KUKA KRL data list: CK1STXXX.dat

&ACCESS RVP
&REL 2
&PARAM EDITMASK = *
DEFDAT  CK1STXXX
;FOLD EXTERNAL DECLARATIONS;%{PE}%MKUKATPBASIS,%CEXT,%VCOMMON,%P
;FOLD BASISTECH EXT;%{PE}%MKUKATPBASIS,%CEXT,%VEXT,%P
EXT  BAS (BAS_COMMAND  :IN,REAL  :IN )
DECL INT SUCCESS
;ENDFOLD (BASISTECH EXT)
;FOLD USER EXT;%{E}%MKUKATPUSER,%CEXT,%VEXT,%P
;Make here your modifications

;ENDFOLD (USER EXT)
;ENDFOLD (EXTERNAL DECLARATIONS)
DECL E6POS XTag7={X -521.268,Y 1581.23206,Z 8.80100,A 49.4600,B 19.4680,C 176.878,S 6,T 59,E1 0.0,E2 0.0,E3 0.0,E4 0.0,E5 0.0,E6 0.0}
DECL FDAT FTag7={TOOL_NO 1,BASE_NO 0,IPO_FRAME #BASE}
DECL PDAT PPDAT1={VEL 80.0000,ACC 100.000,APO_DIST 0.0}
DECL E6POS XTag1={X -521.268,Y 1620.44702,Z -535.910,A 49.4600,B 19.4680,C 176.878,S 6,T 59,E1 0.0,E2 0.0,E3 0.0,E4 0.0,E5 0.0,E6 0.0}
DECL FDAT FTag1={TOOL_NO 1,BASE_NO 0,IPO_FRAME #BASE}
DECL PDAT PPDAT2={VEL 80.0000,ACC 100.000,APO_DIST 100.000}
DECL E6POS XTag2={X -534.322,Y 1875.80,Z -416.009,A 69.9700,B -0.00600000,C 179.993,S 6,T 59,E1 0.0,E2 0.0,E3 0.0,E4 0.0,E5 0.0,E6 0.0}
DECL FDAT FTag2={TOOL_NO 1,BASE_NO 0,IPO_FRAME #BASE}
DECL PDAT PPDAT3={VEL 80.0000,ACC 100.000,APO_DIST 50.0000}
DECL E6POS XTag3={X -534.339,Y 1875.79297,Z -303.179,A 69.9700,B -0.00600000,C 179.993,S 6,T 59,E1 0.0,E2 0.0,E3 0.0,E4 0.0,E5 0.0,E6 0.0}
DECL FDAT FTag3={TOOL_NO 1,BASE_NO 0,IPO_FRAME #BASE}
DECL LDAT LCPDAT1={VEL 0.800000,ACC 100.000,APO_DIST 0.0,APO_FAC 50.0000}
DECL E6POS XTag4={X -534.322,Y 1875.80,Z -416.008,A 69.9700,B -0.00600000,C 179.993,S 6,T 59,E1 0.0,E2 0.0,E3 0.0,E4 0.0,E5 0.0,E6 0.0}
DECL FDAT FTag4={TOOL_NO 1,BASE_NO 0,IPO_FRAME #BASE}
DECL E6POS XTag6={X -421.378204,Y 1411.53516,Z 1878.25,A 56.5646362,B -42.1560,C -128.914,S 6,T 59,E1 0.0,E2 0.0,E3 0.0,E4 0.0,E5 0.0,E6 0.0}
DECL FDAT FTag6={TOOL_NO 1,BASE_NO 0,IPO_FRAME #BASE}
DECL E6POS XTag8={X 942.170,Y 229.415,Z 2855.12793,A -70.4350,B -53.4550,C -81.9820,S 6,T 59,E1 0.0,E2 0.0,E3 0.0,E4 0.0,E5 0.0,E6 0.0}
DECL FDAT FTag8={TOOL_NO 1,BASE_NO 0,IPO_FRAME #BASE}
DECL BASIS_SUGG_T LAST_BASIS={POINT1[] "P1                      ",POINT2[] "P1                      ",CP_PARAMS[] "CPDAT0                  ",PTP_PARAMS[] "PDAT4                   ",CONT[] "                        ",CP_VEL[] "2.0                     ",PTP_VEL[] "80                      ",SYNC_PARAMS[] "SYNCDAT                 ",SPL_NAME[] "S0                      ",A_PARAMS[] "ADAT0                   "}
DECL E6POS XP1={X -653.922058,Y 1817.52954,Z 625.444458,A 72.8232,B -0.974476874,C -162.530731,S 6,T 59,E1 0.0,E2 0.0,E3 0.0,E4 0.0,E5 0.0,E6 0.0}
DECL FDAT FP1={TOOL_NO 1,BASE_NO 0,IPO_FRAME #BASE,POINT2[] " ",TQ_STATE FALSE}
DECL PDAT PPDAT4={VEL 100.000,ACC 100.000,APO_DIST 100.000,GEAR_JERK 50.0000,EXAX_IGN 0}
ENDDAT
